// TIA Portal V18 export
VAR_GLOBAL   // PLC tag table "Default tag table"
   convRight AT %I0.0 : Bool;
   convLeft AT %I0.1 : Bool;
   manualMode AT %Q0.2 : Bool;
   automaticMode AT %Q0.3 : Bool;
END_VAR
